VAR_GLOBAL CONSTANT
	MAX_CLIENT_CONNECTIONS					: UDINT(1..20) := 5;
	PLCPRJ_BUFFER_SIZE						: UDINT := 1000;(* Max. internal fifo/receiver buffer size *)

(*	PLCPRJ_CLIENT_SEND_CYCLE_TIME			: TIME := T#1S; not used at server side *)
	PLCPRJ_RECEIVE_POLLING_TIME				: TIME := T#100MS;
	PLCPRJ_RECEIVE_TIMEOUT					: TIME := T#50S;

	(* Some project specific error codes *)
	PLCPRJ_ERROR_RECEIVE_TIMEOUT			: UDINT := 16#8101;(* Receive timeout *)
	PLCPRJ_ERROR_SENDFIFO_OVERFLOW			: UDINT := 16#8102;(* Send fifo overflow *)
	PLCPRJ_ERROR_RECFIFO_OVERFLOW			: UDINT := 16#8103;(* Receive fifo overflow *)
END_VAR

(* stored: Version 1.1.0.1
   GVL Global_Variables: Id {36b40b87-3807-47c7-adfa-1b692e43fe51} *)
